(* CoDeSys 2.3.9.59 project: Pack_sorter.pro *)
(* Libraries: C:\Program Files (x86)\Common Files\CAA-Targets\Eaton Automation\V2.3.9 SP8\Lib_EC4P-200\SysLibSockets.lib, Standard.lib, SYSLIBCALLBACK.LIB, ModbusTCP.lib 14.11.23 20:05:20 *)

(* PLC configuration (modules and I/O channels)
I1 AT %IX0.0 [LocalBitInput] Input I1
I2 AT %IX0.1 [LocalBitInput] Input I2
I3 AT %IX0.2 [LocalBitInput] Input I3
I4 AT %IX0.3 [LocalBitInput] Input I4
I5 AT %IX0.4 [LocalBitInput] Input I5
I6 AT %IX0.5 [LocalBitInput] Input I6
I7 AT %IX0.6 [LocalBitInput] Input I7
I8 AT %IX0.7 [LocalBitInput] Input I8
I9 AT %IX1.0 [LocalBitInput] Input I9
I10 AT %IX1.1 [LocalBitInput] Input I10
I11 AT %IX1.2 [LocalBitInput] Input I11
I12 AT %IX1.3 [LocalBitInput] Input I12
I13 AT %IX1.4 [LocalDiagInput] Diagnostic Input I13
I14 AT %IX1.5 [LocalDiagInput] Diagnostic Input I14
I15 AT %IX1.6 [LocalDiagInput] Diagnostic Input I15
I16 AT %IX1.7 [LocalDiagInput] Diagnostic Input I16
I7_Analog AT %IW2 [LocalAnalogIn] Input I7, 10Bit, 0-10VDC
I8_Analog AT %IW4 [LocalAnalogIn] Input I8, 10Bit, 0-10VDC
I11_Analog AT %IW6 [LocalAnalogIn] Input I11, 10Bit, 0-10VDC
I12_Analog AT %IW8 [LocalAnalogIn] Input I12, 10Bit, 0-10VDC
Transistor Outputs [EC4P_TOutputs] node 0, in %IB10 out %QB0
  Q1 AT %QX0.0 [LocalBitOutput] Transistor-Output Q1
  Q2 AT %QX0.1 [LocalBitOutput] Transistor-Output Q2
  Q3 AT %QX0.2 [LocalBitOutput] Transistor-Output Q3
  Q4 AT %QX0.3 [LocalBitOutput] Transistor-Output Q4
  Q5 AT %QX0.4 [LocalBitOutput] Transistor-Output Q5
  Q6 AT %QX0.5 [LocalBitOutput] Transistor-Output Q6
  Q7 AT %QX0.6 [LocalBitOutput] Transistor-Output Q7
  Q8 AT %QX0.7 [LocalBitOutput] Transistor-Output Q8
QA1 AT %QW2 [LocalAnalogOut] 10Bit, 0-10VDC Output
No Keys [EC4P_NoKeys] node 2, in %IB10 out %QB4
No Counter [EC4P_NoCounter] node 3, in %IB10 out %QB4
Extension [EC4P_Extension] node 1, in %IB10 out %QB4
  No Extension [EC4P_NoExtension] node 0, in %IB10 out %QB4
*)

(* Global variable list: Global_Variables *)
VAR_GLOBAL
	registers :ARRAY [0..MB_MAXDATAWORDVALUE] OF WORD;
	zdalne_wejscia: ARRAY [0..4] OF WORD;
	zdalne_wyjscia: ARRAY [0..4] OF WORD;
	IZ: ARRAY [0..15] OF BOOL; (*zdalne wejscia cyfrowe*)
	QZ: ARRAY [0..15] OF BOOL; (*zdalne wyjscia cyfrowe*)
	(*valveFillSetpoint:WORD:=27648;
	valveDischargeSetpoint:WORD:=6000;
	pumpBusy:BOOL;
	systemStarted:BOOL:=FALSE;*)
END_VAR

(* Data type *)
TYPE tank :
STRUCT

	levelSensor: REAL;
	flowDischargeSensor:REAL;

	levelSetpoint:REAL:=80;
	levelLow:REAL:=60;

	valveFillAM:BOOL;
	valveFillAuto:BOOL;
	valveFillMan:BOOL;
	valveFillStart:BOOL;

	valveDischargeAM:BOOL;
	valveDischargeAuto:BOOL;
	valveDischargeMan:BOOL;
	valveDischargeStart:BOOL;

	valveFillOutput:WORD;
	valveDischargeOutput:WORD;

	FillStarted:BOOL;

	levelAlarmH:BOOL;
	levelAlarmL:BOOL;
	dischargeFlowAlarm:BOOL;
	generalFault:BOOL;

END_STRUCT
END_TYPE

(* POU PLC_PRG, LD *)
PROGRAM PLC_PRG
VAR
	max_count: INT := 100;
	SHORT_LINE: WORD := 0;
	MEDIUM_LINE: WORD := 1;
	LONG_LINE: WORD := 2;

	line_size0: WORD := 2;
	line_size1: WORD := 1;
	line_size2: WORD := 0;

	delay_emit_time: TIME := t#4s;
	ping1_on_time: TIME := t#4s;
	ping2_on_time: TIME := t#4s;
	ping3_on_time: TIME := t#4s;

	line1_time: TIME := t#6s;
	line2_time: TIME := t#6s;
	line3_time: TIME := t#5s;
	line4_time: TIME := t#6s;

	delay_ping1:  TIME := t#2s;
	delay_ping2: TIME := t#3s;
	delay_ping3: TIME := t#2s;

	destructor_time: TIME := t#5s;

	run: BOOL;
	pack_reset: BOOL;

	pack_detect: size_detect;
	new_size: WORD;
	new_pack_trig: BOOL;
	size0_count: WORD;
	size1_count: WORD;
	size2_count: WORD;

	self_emit: TON;

	pack_tracker_line1: pack_tracker;
	pack_tracker_line2: pack_tracker;
	ping1_stack_down: BOOL;
	ping2_stack_down: BOOL;

	prev_pack_line1: WORD;
	curr_pack_line1: WORD;
	prev_pack_line2: WORD;
	curr_pack_line2: WORD;

	line1_control: line_control;
	ping1_control: ping_control;
	ping1_trig: BOOL;
	ping1_size_fcn: BOOL;
	ping1_validation: ping_valid_fcn;
	ping1_enabled: BOOL;

	line2_control: line_control;
	ping2_control: ping_control1;
	ping2_trig: BOOL;
	ping2_enabled: BOOL;


	line3_control: line_control;
	ping3_control: ping_control;
	ping3_trig: BOOL;
	ping3_enable: BOOL;

	line4_control: line_control;

	destructor_line1: TOF;
	destructor_line2: TOF;
	destructor_line4: TOF;

	size0_ctu: CTU;
	size1_ctu: CTU;
	size2_ctu: CTU;
	size0: BOOL;
	size1: BOOL;
	size2: BOOL;
	emit: BOOL;
	destruct1: BOOL;
	destruct2: BOOL;
	emit_trig: F_TRIG;
	delay_emit: TOF;
	emit_tp: TOF;
	em: R_TRIG;
	p1_a, p1_b, p1_c: BOOL;
	p1_va, p1_vb, p1_vc: BOOL;
	p2_a, p2_b, p2_c: BOOL;
	p2_va, p2_vb, p2_vc: BOOL;
	p3_a, p3_b, p3_c: BOOL;
	p3_va, p3_vb, p3_vc: BOOL;

	size0_butt: button_control;
	size1_butt: button_control;
	size2_butt: button_control;
	stack_down_delay: TOF;
	prolonged_stack_down: BOOL;
	ping1_stack_delay: TOF;
	ping1_stack: BOOL;
	nowy: TP;
	init: BOOL;
	init_val: R_TRIG;
	init_trig: R_TRIG;
	default_values: R_TRIG;
END_VAR
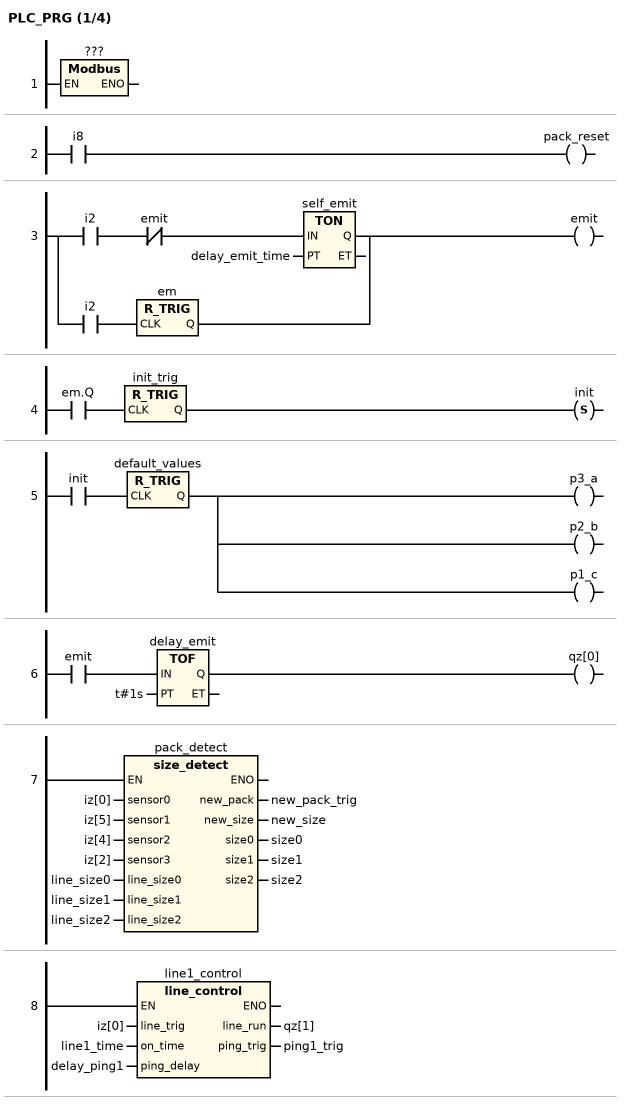
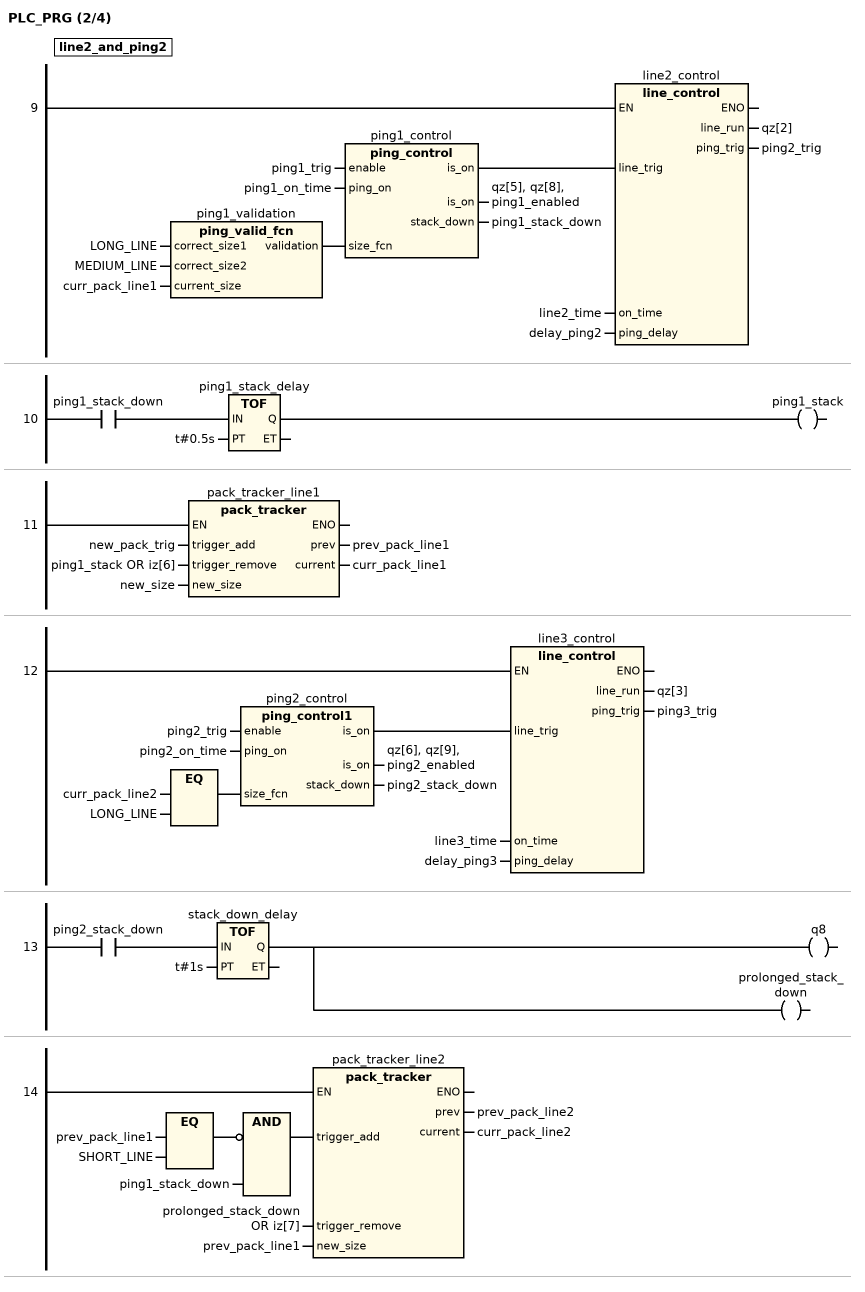
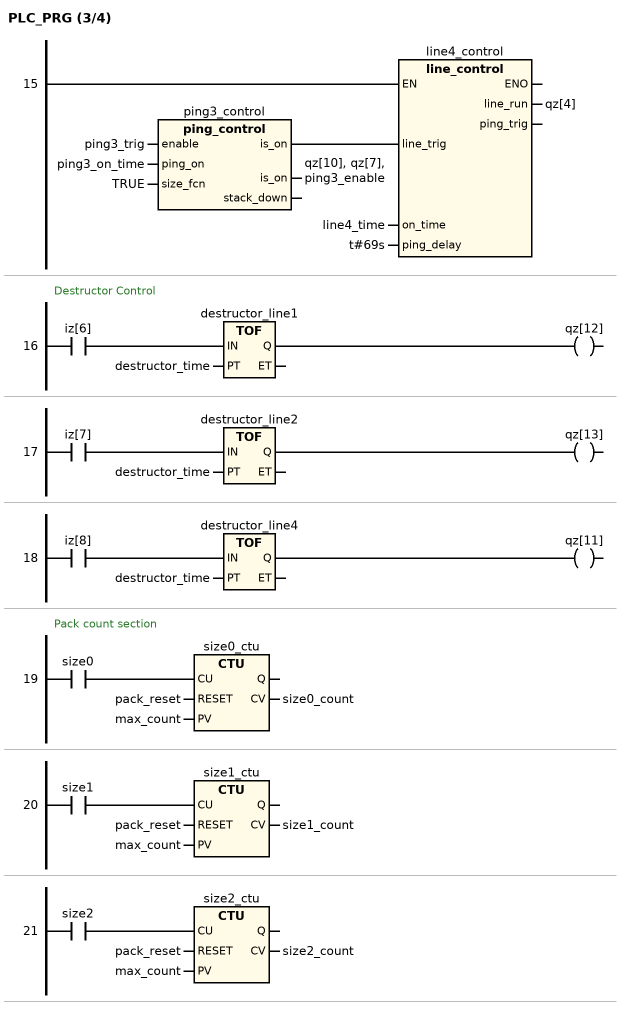
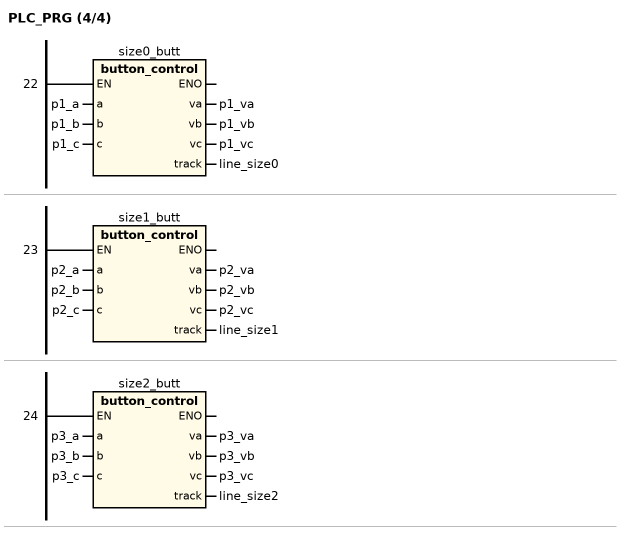
_LD_ (* Ladder Diagram *)
NETWORK 1
	*
		EN --- ???:Modbus()
NETWORK 2
	[i8] --- (pack_reset)
NETWORK 3
	{ [i2] - [/emit] - self_emit:TON(IN: *, PT: delay_emit_time) | [i2] - em:R_TRIG(CLK: *) } --- (emit)
NETWORK 4
	[em.Q] - init_trig:R_TRIG(CLK: *) --- (S init)
NETWORK 5
	[init] - default_values:R_TRIG(CLK: *) --- (p3_a) (p2_b) (p1_c)
NETWORK 6
	[emit] - delay_emit:TOF(IN: *, PT: t#1s) --- (qz[0])
NETWORK 7
	*
		EN --- pack_detect:size_detect(sensor0: iz[0], sensor1: iz[5], sensor2: iz[4], sensor3: iz[2], line_size0: line_size0, line_size1: line_size1, line_size2: line_size2, new_size => new_size, size0 => size0, size1 => size1, size2 => size2) => new_pack_trig
NETWORK 8
	*
		EN --- line1_control:line_control(line_trig: iz[0], on_time: line1_time, ping_delay: delay_ping1, ping_trig => ping1_trig) => qz[1]
NETWORK 9 line2_and_ping2:
	*
		EN --- line2_control:line_control(line_trig: <ping1_control:ping_control(enable: ping1_trig, ping_on: ping1_on_time, size_fcn: ping1_validation:ping_valid_fcn(correct_size1: LONG_LINE, correct_size2: MEDIUM_LINE, current_size: curr_pack_line1), stack_down => ping1_stack_down) => qz[5], qz[8], ping1_enabled>, on_time: line2_time, ping_delay: delay_ping2, ping_trig => ping2_trig) => qz[2]
NETWORK 10
	[ping1_stack_down] - ping1_stack_delay:TOF(IN: *, PT: t#0.5s) --- (ping1_stack)
NETWORK 11
	*
		EN --- pack_tracker_line1:pack_tracker(trigger_add: new_pack_trig, trigger_remove: ping1_stack OR iz[6], new_size: new_size, current => curr_pack_line1) => prev_pack_line1
NETWORK 12
	*
		EN --- line3_control:line_control(line_trig: <ping2_control:ping_control1(enable: ping2_trig, ping_on: ping2_on_time, size_fcn: EQ(curr_pack_line2, LONG_LINE), stack_down => ping2_stack_down) => qz[6], qz[9], ping2_enabled>, on_time: line3_time, ping_delay: delay_ping3, ping_trig => ping3_trig) => qz[3]
NETWORK 13
	[ping2_stack_down] - stack_down_delay:TOF(IN: *, PT: t#1s) --- (q8) (prolonged_stack_down)
NETWORK 14
	*
		EN --- pack_tracker_line2:pack_tracker(trigger_add: AND(NOT EQ(prev_pack_line1, SHORT_LINE), ping1_stack_down), trigger_remove: prolonged_stack_down OR iz[7], new_size: prev_pack_line1, current => curr_pack_line2) => prev_pack_line2
NETWORK 15
	*
		EN --- line4_control:line_control(line_trig: <ping3_control:ping_control(enable: ping3_trig, ping_on: ping3_on_time, size_fcn: TRUE) => qz[10], qz[7], ping3_enable>, on_time: line4_time, ping_delay: t#69s) => qz[4]
NETWORK 16 (* Destructor Control *)
	[iz[6]] - destructor_line1:TOF(IN: *, PT: destructor_time) --- (qz[12])
NETWORK 17
	[iz[7]] - destructor_line2:TOF(IN: *, PT: destructor_time) --- (qz[13])
NETWORK 18
	[iz[8]] - destructor_line4:TOF(IN: *, PT: destructor_time) --- (qz[11])
NETWORK 19 (* Pack count section *)
	[size0] - size0_ctu:CTU(CU: *, RESET: pack_reset, PV: max_count, CV => size0_count)
NETWORK 20
	[size1] - size1_ctu:CTU(CU: *, RESET: pack_reset, PV: max_count, CV => size1_count)
NETWORK 21
	[size2] - size2_ctu:CTU(CU: *, RESET: pack_reset, PV: max_count, CV => size2_count)
NETWORK 22
	*
		EN --- size0_butt:button_control(a: p1_a, b: p1_b, c: p1_c, vb => p1_vb, vc => p1_vc, track => line_size0) => p1_va
NETWORK 23
	*
		EN --- size1_butt:button_control(a: p2_a, b: p2_b, c: p2_c, vb => p2_vb, vc => p2_vc, track => line_size1) => p2_va
NETWORK 24
	*
		EN --- size2_butt:button_control(a: p3_a, b: p3_b, c: p3_c, vb => p3_vb, vc => p3_vc, track => line_size2) => p3_va
_END_LD_
(* the same logic as Structured Text *)
(* Network 1: see the listing above *)
(* Network 2 *)
pack_reset := i8;
(* Network 3 *)
self_emit(IN := i2 AND NOT emit, PT := delay_emit_time);
em(CLK := i2);
emit := self_emit.Q OR em.Q;
(* Network 4 *)
init_trig(CLK := em.Q);
IF init_trig.Q THEN init := TRUE; END_IF;
(* Network 5 *)
default_values(CLK := init);
p3_a := default_values.Q;
p2_b := default_values.Q;
p1_c := default_values.Q;
(* Network 6 *)
delay_emit(IN := emit, PT := t#1s);
qz[0] := delay_emit.Q;
(* Network 7 *)
pack_detect(sensor0 := iz[0], sensor1 := iz[5], sensor2 := iz[4], sensor3 := iz[2], line_size0 := line_size0, line_size1 := line_size1, line_size2 := line_size2);
new_size := pack_detect.new_size;
size0 := pack_detect.size0;
size1 := pack_detect.size1;
size2 := pack_detect.size2;
new_pack_trig := pack_detect.new_pack;
(* Network 8 *)
line1_control(line_trig := iz[0], on_time := line1_time, ping_delay := delay_ping1);
ping1_trig := line1_control.ping_trig;
qz[1] := line1_control.line_run;
(* Network 9: see the listing above *)
(* Network 10 *)
ping1_stack_delay(IN := ping1_stack_down, PT := t#0.5s);
ping1_stack := ping1_stack_delay.Q;
(* Network 11 *)
pack_tracker_line1(trigger_add := new_pack_trig, trigger_remove := ping1_stack OR iz[6], new_size := new_size);
curr_pack_line1 := pack_tracker_line1.current;
prev_pack_line1 := pack_tracker_line1.prev;
(* Network 12: see the listing above *)
(* Network 13 *)
stack_down_delay(IN := ping2_stack_down, PT := t#1s);
q8 := stack_down_delay.Q;
prolonged_stack_down := stack_down_delay.Q;
(* Network 14 *)
pack_tracker_line2(trigger_add := NOT (prev_pack_line1 = SHORT_LINE) AND ping1_stack_down, trigger_remove := prolonged_stack_down OR iz[7], new_size := prev_pack_line1);
curr_pack_line2 := pack_tracker_line2.current;
prev_pack_line2 := pack_tracker_line2.prev;
(* Network 15: see the listing above *)
(* Network 16 *)
destructor_line1(IN := iz[6], PT := destructor_time);
qz[12] := destructor_line1.Q;
(* Network 17 *)
destructor_line2(IN := iz[7], PT := destructor_time);
qz[13] := destructor_line2.Q;
(* Network 18 *)
destructor_line4(IN := iz[8], PT := destructor_time);
qz[11] := destructor_line4.Q;
(* Network 19 *)
size0_ctu(CU := size0, RESET := pack_reset, PV := max_count);
size0_count := size0_ctu.CV;
(* Network 20 *)
size1_ctu(CU := size1, RESET := pack_reset, PV := max_count);
size1_count := size1_ctu.CV;
(* Network 21 *)
size2_ctu(CU := size2, RESET := pack_reset, PV := max_count);
size2_count := size2_ctu.CV;
(* Network 22 *)
size0_butt(a := p1_a, b := p1_b, c := p1_c);
p1_vb := size0_butt.vb;
p1_vc := size0_butt.vc;
line_size0 := size0_butt.track;
p1_va := size0_butt.va;
(* Network 23 *)
size1_butt(a := p2_a, b := p2_b, c := p2_c);
p2_vb := size1_butt.vb;
p2_vc := size1_butt.vc;
line_size1 := size1_butt.track;
p2_va := size1_butt.va;
(* Network 24 *)
size2_butt(a := p3_a, b := p3_b, c := p3_c);
p3_vb := size2_butt.vb;
p3_vc := size2_butt.vc;
line_size2 := size2_butt.track;
p3_va := size2_butt.va;
END_PROGRAM

(* POU size_detect, ST *)
FUNCTION_BLOCK size_detect
VAR_INPUT
	(*  iz[0] - s0; iz[5] - s1; iz[4]; s2-  iz[2] *)
	sensor0, sensor1, sensor2, sensor3: BOOL;
	line_size0, line_size1, line_size2: WORD;
END_VAR
VAR_OUTPUT
	new_pack: BOOL;
	new_size: WORD;
	size0, size1, size2: BOOL;
END_VAR
VAR
	size0_trg, reset_trg, size2_trg: R_TRIG;
	size0_det: BOOL := FALSE;
END_VAR
size0_trg(CLK := sensor0);
size2_trg(CLK := sensor2);
reset_trg(CLK := sensor3);

IF size0_trg.Q AND sensor1 THEN
	new_size := line_size0;
	size0  := TRUE;
	size1 := FALSE;
	size2 := FALSE;
	size0_det := TRUE;

	new_pack := TRUE;
ELSIF size2_trg.Q AND NOT size0_det  THEN
	IF sensor3 THEN
		new_size := line_size1;
		size1  := TRUE;
		size0 := FALSE;
		size2 := FALSE;
		size0_det := FALSE;

		new_pack := TRUE;
	ELSE
		new_size := line_size2;
		size2  := TRUE;
		size1 := FALSE;
		size0 := FALSE;
		size0_det := FALSE;

		new_pack := TRUE;
	END_IF;
ELSIF reset_trg.Q THEN
	size0_det := FALSE;
	size1 := FALSE;
	size1 := FALSE;
	size0 := FALSE;
ELSE
	new_pack := FALSE;
	size1 := FALSE;
	size1 := FALSE;
	size0 := FALSE;
END_IF;
END_FUNCTION_BLOCK

(* POU pack_tracker, ST *)
FUNCTION_BLOCK pack_tracker
VAR_INPUT
	trigger_add: BOOL;
	trigger_remove: BOOL;
	new_size: WORD;
END_VAR
VAR_OUTPUT
	prev: WORD := 255;
	current: WORD := 255;
END_VAR
VAR
	stack_size: INT := 6;
	stack : ARRAY [1..6] OF WORD;
	stack_init: BOOL := TRUE;

	stack_up_trig: R_TRIG;
	stack_down_trig: R_TRIG;
	i: INT;
END_VAR
stack_up_trig(CLK := trigger_add);
stack_down_trig(CLK := trigger_remove);

IF stack_init THEN
	FOR i :=1 TO stack_size DO
		stack[i] := 255;
	END_FOR;
	stack_init := FALSE;
END_IF;

IF stack_down_trig.Q THEN
	prev := stack[1];
	FOR i := 1 TO stack_size-1 DO
		IF stack[i] = 255 THEN
			EXIT;
		END_IF;

		stack[i] := stack[i+1];
	END_FOR;
	current := stack[1];
END_IF;

IF stack_up_trig.Q THEN
	FOR i := 1	 TO stack_size-1 DO
		IF stack[i] = 255 THEN
			stack[i] := new_size;
			IF i = 1 THEN
				current := new_size;
			END_IF;

			EXIT;
		END_IF;
	END_FOR;
END_IF;
END_FUNCTION_BLOCK

(* POU line_control, LD *)
FUNCTION_BLOCK line_control
VAR_INPUT
	line_trig: BOOL;
	on_time: TIME;
	ping_delay: TIME;
END_VAR
VAR_OUTPUT
	line_run: BOOL;
	ping_trig: BOOL;
END_VAR
VAR
	line_enable_trig: R_TRIG;
	line_on: BOOL;
	ping_timer: TON;
	line_run_timer: TOF;
	ping_off: BOOL;
	timing_error: BOOL;

	ping_delay_timer: TP;
	ping_trigger: F_TRIG;
END_VAR
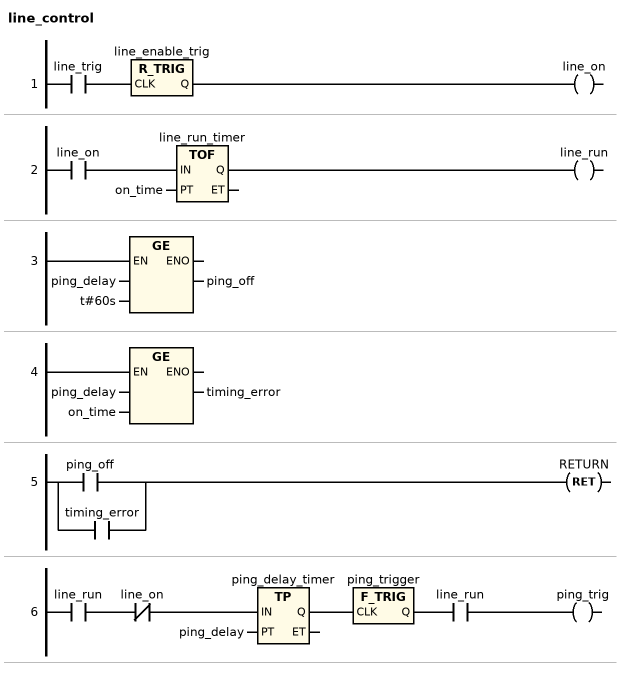
_LD_ (* Ladder Diagram *)
NETWORK 1
	[line_trig] - line_enable_trig:R_TRIG(CLK: *) --- (line_on)
NETWORK 2
	[line_on] - line_run_timer:TOF(IN: *, PT: on_time) --- (line_run)
NETWORK 3
	*
		EN --- GE(ping_delay, t#60s) => ping_off
NETWORK 4
	*
		EN --- GE(ping_delay, on_time) => timing_error
NETWORK 5
	{ [ping_off] | [timing_error] } --- <RETURN>
NETWORK 6
	[line_run] - [/line_on] - ping_delay_timer:TP(IN: *, PT: ping_delay) - ping_trigger:F_TRIG(CLK: *) - [line_run] --- (ping_trig)
_END_LD_
(* the same logic as Structured Text *)
(* Network 1 *)
line_enable_trig(CLK := line_trig);
line_on := line_enable_trig.Q;
(* Network 2 *)
line_run_timer(IN := line_on, PT := on_time);
line_run := line_run_timer.Q;
(* Network 3 *)
ping_off := ping_delay >= t#60s;
(* Network 4 *)
timing_error := ping_delay >= on_time;
(* Network 5 *)
IF ping_off OR timing_error THEN RETURN; END_IF;
(* Network 6 *)
ping_delay_timer(IN := line_run AND NOT line_on, PT := ping_delay);
ping_trigger(CLK := ping_delay_timer.Q);
ping_trig := ping_trigger.Q AND line_run;
END_FUNCTION_BLOCK

(* POU ping_control, LD *)
FUNCTION_BLOCK ping_control
VAR_INPUT
	enable: BOOL;
	ping_on: TIME;
	size_fcn: BOOL;
END_VAR
VAR_OUTPUT
	is_on: BOOL;
	stack_down: BOOL;
END_VAR
VAR
	start_time: R_TRIG;
	turn_on: BOOL;
	delay_timer: TOF;
	size: BOOL;
	helper_counter: CTUD;
	odd_pack: BOOL;
	even_pack: BOOL;
	even_pack_timer: TOF;
	odd_pack_timer: TOF;
	stack_down_trig: F_TRIG;
	stack_down_odd: BOOL;
	stack_down_odd_trig: F_TRIG;
	stack_down_even_trig: F_TRIG;
	stack_down_even: BOOL;
	odd_timer_trig: F_TRIG;
	even_timer_trig: F_TRIG;
	cu_en: BOOL;
	cd_en: BOOL;
	od_tp: TP;
	ev_tp: TP;
END_VAR
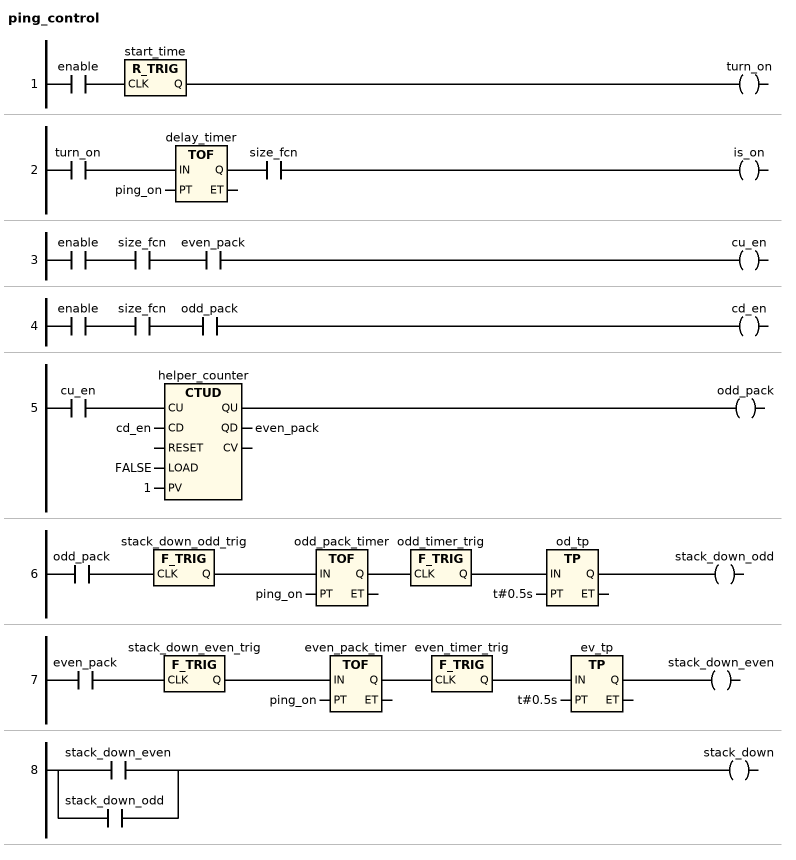
_LD_ (* Ladder Diagram *)
NETWORK 1
	[enable] - start_time:R_TRIG(CLK: *) --- (turn_on)
NETWORK 2
	[turn_on] - delay_timer:TOF(IN: *, PT: ping_on) - [size_fcn] --- (is_on)
NETWORK 3
	[enable] - [size_fcn] - [even_pack] --- (cu_en)
NETWORK 4
	[enable] - [size_fcn] - [odd_pack] --- (cd_en)
NETWORK 5
	[cu_en] - helper_counter:CTUD(CU: *, CD: cd_en, RESET: , LOAD: FALSE, PV: 1, QD => even_pack) --- (odd_pack)
NETWORK 6
	[odd_pack] - stack_down_odd_trig:F_TRIG(CLK: *) - odd_pack_timer:TOF(IN: *, PT: ping_on) - odd_timer_trig:F_TRIG(CLK: *) - od_tp:TP(IN: *, PT: t#0.5s) --- (stack_down_odd)
NETWORK 7
	[even_pack] - stack_down_even_trig:F_TRIG(CLK: *) - even_pack_timer:TOF(IN: *, PT: ping_on) - even_timer_trig:F_TRIG(CLK: *) - ev_tp:TP(IN: *, PT: t#0.5s) --- (stack_down_even)
NETWORK 8
	{ [stack_down_even] | [stack_down_odd] } --- (stack_down)
_END_LD_
(* the same logic as Structured Text *)
(* Network 1 *)
start_time(CLK := enable);
turn_on := start_time.Q;
(* Network 2 *)
delay_timer(IN := turn_on, PT := ping_on);
is_on := delay_timer.Q AND size_fcn;
(* Network 3 *)
cu_en := enable AND size_fcn AND even_pack;
(* Network 4 *)
cd_en := enable AND size_fcn AND odd_pack;
(* Network 5: see the listing above *)
(* Network 6 *)
stack_down_odd_trig(CLK := odd_pack);
odd_pack_timer(IN := stack_down_odd_trig.Q, PT := ping_on);
odd_timer_trig(CLK := odd_pack_timer.Q);
od_tp(IN := odd_timer_trig.Q, PT := t#0.5s);
stack_down_odd := od_tp.Q;
(* Network 7 *)
stack_down_even_trig(CLK := even_pack);
even_pack_timer(IN := stack_down_even_trig.Q, PT := ping_on);
even_timer_trig(CLK := even_pack_timer.Q);
ev_tp(IN := even_timer_trig.Q, PT := t#0.5s);
stack_down_even := ev_tp.Q;
(* Network 8 *)
stack_down := stack_down_even OR stack_down_odd;
END_FUNCTION_BLOCK

(* POU ping_valid_fcn, LD *)
FUNCTION_BLOCK ping_valid_fcn
VAR_INPUT
	correct_size1, correct_size2: WORD;
	current_size: WORD;
END_VAR
VAR_OUTPUT
	validation: BOOL;
END_VAR
VAR
END_VAR
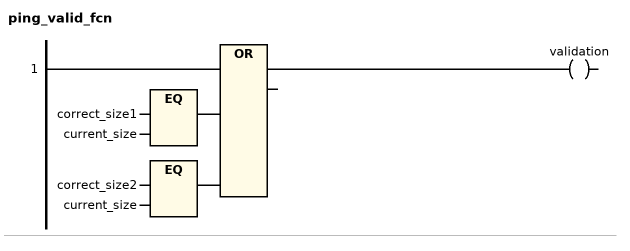
_LD_ (* Ladder Diagram *)
NETWORK 1
	OR(EQ(correct_size1, current_size), EQ(correct_size2, current_size)) --- (validation)
_END_LD_
END_FUNCTION_BLOCK

(* POU ping_control1, LD *)
FUNCTION_BLOCK ping_control1
VAR_INPUT
	enable: BOOL;
	ping_on: TIME;
	size_fcn: BOOL;
END_VAR
VAR_OUTPUT
	is_on: BOOL;
	stack_down: BOOL;
END_VAR
VAR
	start_time: R_TRIG;
	turn_on: BOOL;
	delay_timer: TOF;
	size: BOOL;
	helper_counter: CTUD;
	odd_pack: BOOL;
	even_pack: BOOL;
	even_pack_timer: TOF;
	odd_pack_timer: TOF;
	stack_down_trig: F_TRIG;
	stack_down_odd: BOOL;
	stack_down_odd_trig: F_TRIG;
	stack_down_even_trig: F_TRIG;
	stack_down_even: BOOL;
	odd_timer_trig: F_TRIG;
	even_timer_trig: F_TRIG;
	cu_en: BOOL;
	cd_en: BOOL;
	init: BOOL;
	init_trig: R_TRIG;
	od: TP;
	ev: TP;
END_VAR
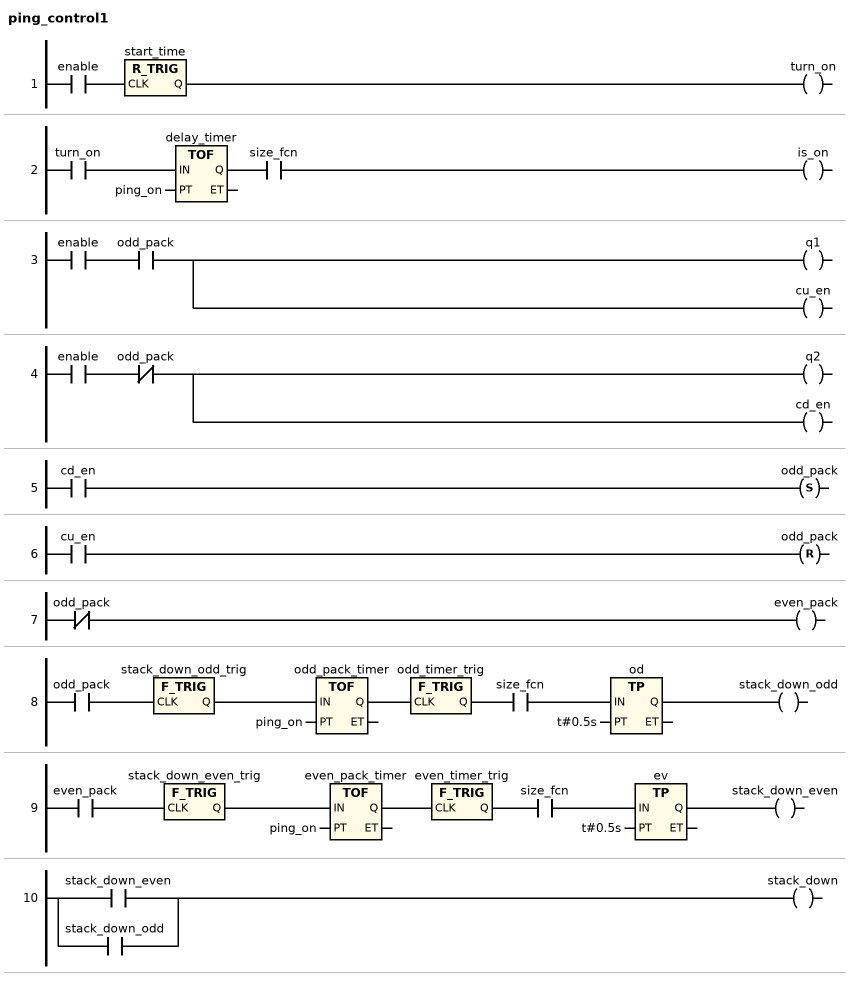
_LD_ (* Ladder Diagram *)
NETWORK 1
	[enable] - start_time:R_TRIG(CLK: *) --- (turn_on)
NETWORK 2
	[turn_on] - delay_timer:TOF(IN: *, PT: ping_on) - [size_fcn] --- (is_on)
NETWORK 3
	[enable] - [odd_pack] --- (q1) (cu_en)
NETWORK 4
	[enable] - [/odd_pack] --- (q2) (cd_en)
NETWORK 5
	[cd_en] --- (S odd_pack)
NETWORK 6
	[cu_en] --- (R odd_pack)
NETWORK 7
	[/odd_pack] --- (even_pack)
NETWORK 8
	[odd_pack] - stack_down_odd_trig:F_TRIG(CLK: *) - odd_pack_timer:TOF(IN: *, PT: ping_on) - odd_timer_trig:F_TRIG(CLK: *) - [size_fcn] - od:TP(IN: *, PT: t#0.5s) --- (stack_down_odd)
NETWORK 9
	[even_pack] - stack_down_even_trig:F_TRIG(CLK: *) - even_pack_timer:TOF(IN: *, PT: ping_on) - even_timer_trig:F_TRIG(CLK: *) - [size_fcn] - ev:TP(IN: *, PT: t#0.5s) --- (stack_down_even)
NETWORK 10
	{ [stack_down_even] | [stack_down_odd] } --- (stack_down)
_END_LD_
(* the same logic as Structured Text *)
(* Network 1 *)
start_time(CLK := enable);
turn_on := start_time.Q;
(* Network 2 *)
delay_timer(IN := turn_on, PT := ping_on);
is_on := delay_timer.Q AND size_fcn;
(* Network 3 *)
q1 := enable AND odd_pack;
cu_en := q1;
(* Network 4 *)
q2 := enable AND NOT odd_pack;
cd_en := q2;
(* Network 5 *)
IF cd_en THEN odd_pack := TRUE; END_IF;
(* Network 6 *)
IF cu_en THEN odd_pack := FALSE; END_IF;
(* Network 7 *)
even_pack := NOT odd_pack;
(* Network 8 *)
stack_down_odd_trig(CLK := odd_pack);
odd_pack_timer(IN := stack_down_odd_trig.Q, PT := ping_on);
odd_timer_trig(CLK := odd_pack_timer.Q);
od(IN := odd_timer_trig.Q AND size_fcn, PT := t#0.5s);
stack_down_odd := od.Q;
(* Network 9 *)
stack_down_even_trig(CLK := even_pack);
even_pack_timer(IN := stack_down_even_trig.Q, PT := ping_on);
even_timer_trig(CLK := even_pack_timer.Q);
ev(IN := even_timer_trig.Q AND size_fcn, PT := t#0.5s);
stack_down_even := ev.Q;
(* Network 10 *)
stack_down := stack_down_even OR stack_down_odd;
END_FUNCTION_BLOCK

(* POU button_control, LD *)
FUNCTION_BLOCK button_control
VAR_INPUT
	a, b, c : BOOL;
END_VAR
VAR_OUTPUT
	va, vb, vc: BOOL;
	track: WORD;
END_VAR
VAR
END_VAR
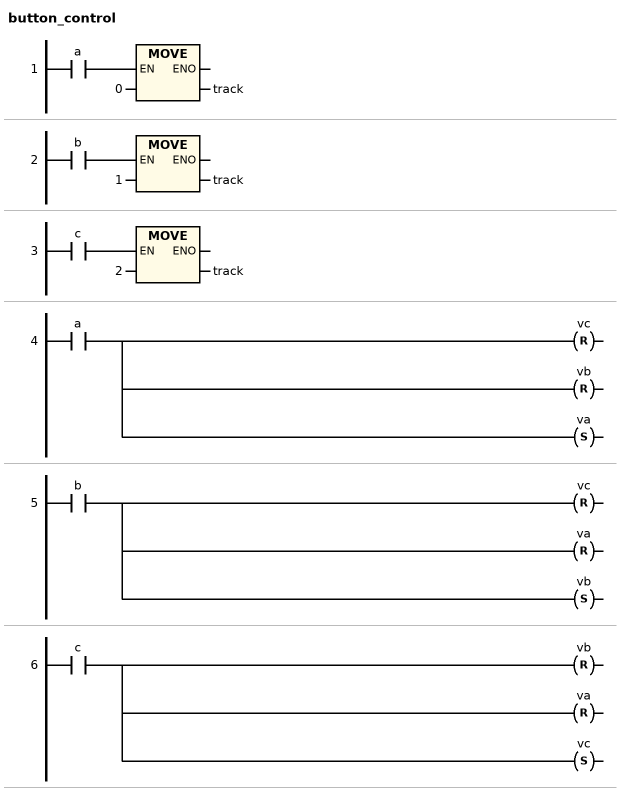
_LD_ (* Ladder Diagram *)
NETWORK 1
	[a]
		EN --- MOVE(0) => track
NETWORK 2
	[b]
		EN --- MOVE(1) => track
NETWORK 3
	[c]
		EN --- MOVE(2) => track
NETWORK 4
	[a] --- (R vc) (R vb) (S va)
NETWORK 5
	[b] --- (R vc) (R va) (S vb)
NETWORK 6
	[c] --- (R vb) (R va) (S vc)
_END_LD_
(* the same logic as Structured Text *)
(* Network 1 *)
IF a THEN
	track := 0;
END_IF;
(* Network 2 *)
IF b THEN
	track := 1;
END_IF;
(* Network 3 *)
IF c THEN
	track := 2;
END_IF;
(* Network 4 *)
IF a THEN vc := FALSE; vb := FALSE; va := TRUE; END_IF;
(* Network 5 *)
IF b THEN vc := FALSE; va := FALSE; vb := TRUE; END_IF;
(* Network 6 *)
IF c THEN vb := FALSE; va := FALSE; vc := TRUE; END_IF;
END_FUNCTION_BLOCK

(* POU Modbus, ST *)
PROGRAM Modbus

VAR
	modbusError: WORD;
	modbusTCP_server:FB_serverModbusTCP;
	FB_mapInputRegister:FB_mapInputRegister;
	FB_mapOutputRegister:FB_mapOutputRegister;
	FB_startSystem:FB_startSystem;
	FB_liveBitMonitor:FB_liveBitMonitor;
	startDischarge: BOOL;
	deviceFault: BOOL;
	faultAcknowledge: BOOL;
	i:SINT;
	stopLight: BOOL;
	voltageLight: BOOL;
	liveBitBitInput: BOOL;
	liveBitBitOutput: BOOL;
	modbusTimeoutError: BOOL;
	copy_zdalne1: copy_zdalne;
END_VAR
(* Modbus server FB *)
modbusTCP_server(ServerID:=255 , ServerPort:=502 , LastError=>modbusError);

(* Mapping input registers to variables *)
copy_zdalne1(EN:=TRUE);

(*FB_mapInputRegister(
	inputHoldingRegister:=registers[0] ,
	bit0=> Q1,
	bit1=> Q2,
	bit2=> Q3,
	bit3=> Q4,
	bit4=> Q5,
	bit5=> Q6 ,
	bit6=> Q7,
	bit7=> Q8,
	bit8=> ,
	bit9=> ,
	bit10=> ,
	bit11=> ,
	bit12=> ,
	bit13=> ,
	bit14=> ,
	bit15=> liveBitBitInput);
*)
FB_mapInputRegister(
	inputHoldingRegister:=registers[0] ,
	bit0=> IZ[0],
	bit1=> IZ[1],
	bit2=> IZ[2],
	bit3=> IZ[3],
	bit4=> IZ[4],
	bit5=> IZ[5] ,
	bit6=> IZ[6],
	bit7=> IZ[7],
	bit8=> IZ[8],
	bit9=> IZ[9],
	bit10=> IZ[10],
	bit11=> IZ[11],
	bit12=> IZ[12],
	bit13=> IZ[13],
	bit14=> IZ[14],
	bit15=> IZ[15]);

(* Modbus liveBit *)
FB_liveBitMonitor(liveBitInput:=liveBitBitInput , liveBitOutput=>liveBitBitOutput , liveBitError=> modbusTimeoutError);

(* Process faults *)


(* Process control *)



(* Fault acknowledge *)



(* Map variables to output registers *)

FB_mapOutputRegister(
	bit0:= QZ[0],
	bit1:= QZ[1],
	bit2:= QZ[2],
	bit3:= QZ[3],
	bit4:= QZ[4],
	bit5:= QZ[5],
	bit6:= QZ[6],
	bit7:= QZ[7],
	bit8:= QZ[8],
	bit9:= QZ[9],
	bit10:= QZ[10],
	bit11:= QZ[11],
	bit12:= QZ[12],
	bit13:= QZ[13],
	bit14:= QZ[14],
	bit15:= QZ[15],
	outputHoldingRegister=>registers[60] );
(*FB_mapOutputRegister(
	bit0:= I1,
	bit1:= I2,
	bit2:= I3,
	bit3:= I4,
	bit4:= I5,
	bit5:= I6,
	bit6:= I7,
	bit7:= I8,
	bit8:= I9,
	bit9:= I10,
	bit10:= I11,
	bit11:= I12,
	bit12:= ,
	bit13:= ,
	bit14:= ,
	bit15:= ,
	outputHoldingRegister=>registers[60] );
*)

qa1:= REGISTERS[1];
registers[61]:=i7_analog;
registers[62]:=i8_analog;

registers[63]:=i11_analog;
registers[64]:=i12_analog;

registers[65]:=0;
registers[66]:=0;

registers[67]:=0;
registers[68]:=0;

registers[119] := registers[119]+1;
END_PROGRAM

(* POU FBs/FB_serverModbusTCP, ST *)
FUNCTION_BLOCK FB_serverModbusTCP
VAR_INPUT
	ServerID:BYTE;
	ServerPort:INT;
END_VAR
VAR_OUTPUT
	LastError:INT;
END_VAR
VAR
	SlaveSetup:MBS_Setup;
	SlavePoll:MBS_Poll;
	SlaveAnswer:MBS_Answer;
	step: USINT :=0;
	i: INT;
END_VAR
CASE step OF
0:	(*Initialisation*)

	SlaveSetup.bUnitIdentifier := ServerID;
	MBS_AcceptAllSubunitIds := TRUE;

	SlaveSetup.wDefaultPort :=ServerPort;
	SlaveSetup.xDefaultPortActive:=TRUE;
	SlaveSetup.xAdditionalPortActive:=FALSE;

	SlaveSetup.xSecureMode:=FALSE;			(*If TRUE only preset IPs are accepted*)
	SlaveSetup.tTimeout:=T#1m;					(*Timeout if no communication with slave established*)
	SlaveSetup(xStrobe:=TRUE);					(*Strobe starts function*)
	IF SlaveSetup.xBusy = FALSE THEN
		SlaveSetup(xstrobe := FALSE);			(*provides falling edge*)
		step := 1 ;
	END_IF;
1:
	SlavePoll(xStrobe:=TRUE);					(*waiting for incomming master commands*)
		IF NOT SlavePoll.xBusy THEN
			step:=2;							(*hint: step 1 & 2 could be merged to accelerate slave handling, if needed*)
			SlavePoll(xStrobe:=FALSE);			(*provides falling edge*)
		END_IF;

2:
	step:= 1;

	IF  SlavePoll.xAvailable = TRUE  THEN

		IF SlavePoll.iErrorCode <> 0 THEN
			LastError := SlavePoll.iErrorCode;									(* provided for error treatment *)
		END_IF;

		CASE SlavePoll.bFunctionCode OF										(* connect accepted pollparameters with answerparameters *)
			16:
				slaveanswer.bFunctionCode:=slavepoll.bFunctionCode;
				slaveanswer.wCount:=slavepoll.wCount;
				slaveanswer.wOffset:=slavepoll.wOffset;
				FOR i := 0 TO slaveanswer.wCount-1 BY 1 DO
					registers[slaveanswer.woffset+i] := slavepoll.warData[i];		(*Write to Data-array*)
				END_FOR;
				slaveanswer.wardata := slavepoll.warData;
			4:
				slaveanswer.bFunctionCode:=slavepoll.bFunctionCode;
				slaveanswer.wCount:=slavepoll.wCount;
				slaveanswer.wOffset:=slavepoll.wOffset;
				FOR i:= 0 TO slaveanswer.wCount-1 BY 1 DO
					slaveanswer.warData[i]:=registers[slavepoll.woffset+i];			(*Read from Data-array*)
				END_FOR
		END_CASE;

		slaveanswer();	(*When Data ready, send answer*)

	END_IF;
END_CASE;
END_FUNCTION_BLOCK

(* POU FBs/FB_mapInputRegister, ST *)
FUNCTION_BLOCK FB_mapInputRegister
VAR_INPUT
	inputHoldingRegister : WORD;
END_VAR
VAR_OUTPUT
	bit0 : BOOL;
	bit1 : BOOL;
	bit2 : BOOL;
	bit3 : BOOL;
	bit4 : BOOL;
	bit5 : BOOL;
	bit6 : BOOL;
	bit7 : BOOL;
	bit8 : BOOL;
	bit9 : BOOL;
	bit10 : BOOL;
	bit11 : BOOL;
	bit12 : BOOL;
	bit13 : BOOL;
	bit14 : BOOL;
	bit15 : BOOL;
END_VAR
VAR
END_VAR
bit0 :=inputHoldingRegister.0;
bit1 :=inputHoldingRegister.1;
bit2 :=inputHoldingRegister.2;
bit3 :=inputHoldingRegister.3;
bit4 :=inputHoldingRegister.4;
bit5 :=inputHoldingRegister.5;
bit6 :=inputHoldingRegister.6;
bit7 :=inputHoldingRegister.7;
bit8 :=inputHoldingRegister.8;
bit9 :=inputHoldingRegister.9;
bit10 :=inputHoldingRegister.10;
bit11 :=inputHoldingRegister.11;
bit12 :=inputHoldingRegister.12;
bit13 :=inputHoldingRegister.13;
bit14 :=inputHoldingRegister.14;
bit15 :=inputHoldingRegister.15;
END_FUNCTION_BLOCK

(* POU FBs/FB_mapOutputRegister, ST *)
FUNCTION_BLOCK FB_mapOutputRegister
VAR_INPUT
	bit0 : BOOL;
	bit1 : BOOL;
	bit2 : BOOL;
	bit3 : BOOL;
	bit4 : BOOL;
	bit5 : BOOL;
	bit6 : BOOL;
	bit7 : BOOL;
	bit8 : BOOL;
	bit9 : BOOL;
	bit10 : BOOL;
	bit11 : BOOL;
	bit12 : BOOL;
	bit13 : BOOL;
	bit14 : BOOL;
	bit15 : BOOL;
END_VAR
VAR_OUTPUT
	outputHoldingRegister : WORD;
END_VAR
VAR
END_VAR
outputHoldingRegister.0:=bit0;
outputHoldingRegister.1:=bit1;
outputHoldingRegister.2:=bit2;
outputHoldingRegister.3:=bit3;
outputHoldingRegister.4:=bit4;
outputHoldingRegister.5:=bit5;
outputHoldingRegister.6:=bit6;
outputHoldingRegister.7:=bit7;
outputHoldingRegister.8:=bit8;
outputHoldingRegister.9:=bit9;
outputHoldingRegister.10:=bit10;
outputHoldingRegister.11:=bit11;
outputHoldingRegister.12:=bit12;
outputHoldingRegister.13:=bit13;
outputHoldingRegister.14:=bit14;
outputHoldingRegister.15:=bit15;
END_FUNCTION_BLOCK

(* POU FBs/FB_startSystem, LD *)
FUNCTION_BLOCK FB_startSystem
VAR_INPUT
	start:BOOL;
	stop:BOOL;
	safety:BOOL;
	reset:BOOL;
	fault:BOOL;
END_VAR
VAR_OUTPUT
	systemStarted:BOOL;
	systemStopLight: BOOL;
	safetyRS: BOOL:=TRUE;
END_VAR
VAR
	TOF_BLINK: TOF;
	TON_BLINK: TON;

END_VAR
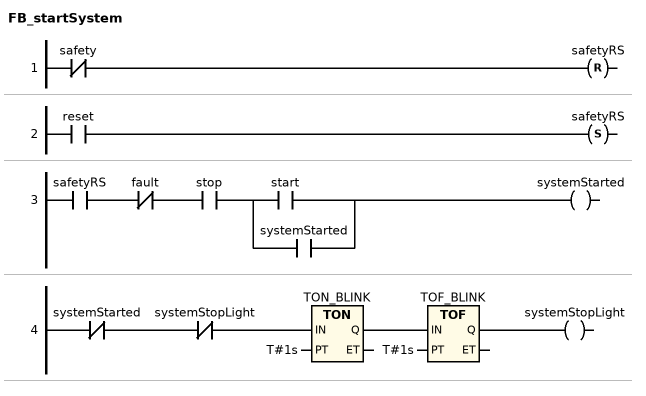
_LD_ (* Ladder Diagram *)
NETWORK 1
	[/safety] --- (R safetyRS)
NETWORK 2
	[reset] --- (S safetyRS)
NETWORK 3
	[safetyRS] - [/fault] - [stop] - { [start] | [systemStarted] } --- (systemStarted)
NETWORK 4
	[/systemStarted] - [/systemStopLight] - TON_BLINK:TON(IN: *, PT: T#1s) - TOF_BLINK:TOF(IN: *, PT: T#1s) --- (systemStopLight)
_END_LD_
(* the same logic as Structured Text *)
(* Network 1 *)
IF NOT safety THEN safetyRS := FALSE; END_IF;
(* Network 2 *)
IF reset THEN safetyRS := TRUE; END_IF;
(* Network 3 *)
systemStarted := safetyRS AND NOT fault AND stop AND (start OR systemStarted);
(* Network 4 *)
TON_BLINK(IN := NOT systemStarted AND NOT systemStopLight, PT := T#1s);
TOF_BLINK(IN := TON_BLINK.Q, PT := T#1s);
systemStopLight := TOF_BLINK.Q;
END_FUNCTION_BLOCK

(* POU FBs/FB_liveBitMonitor, ST *)
FUNCTION_BLOCK FB_liveBitMonitor
VAR_INPUT
	liveBitInput:BOOL;
END_VAR
VAR_OUTPUT
	liveBitOutput:BOOL;
	liveBitError:BOOL;
END_VAR
VAR
	inputR_TRIG: R_TRIG;
	liveBitTON: TON;
END_VAR
inputR_TRIG(CLK:=liveBitInput , Q=> );

liveBitTON(IN:= NOT inputR_TRIG.Q , PT:= T#3s , Q=> , ET=> );

IF liveBitTON.Q THEN
	liveBitError:=TRUE;
END_IF;
IF inputR_TRIG.Q THEN
	liveBitError:=FALSE;
END_IF

liveBitOutput := liveBitInput;
END_FUNCTION_BLOCK

(* POU FBs/copy_zdalne, ST *)
FUNCTION_BLOCK copy_zdalne
VAR_INPUT
	EN:BOOL;
END_VAR
VAR_OUTPUT
END_VAR
VAR
	k:INT;
END_VAR
(*FOR k:=0 TO 15 BY 1 DO
	zdalne_wyjscia[0].k := QZ[k];
END_FOR*)
IF EN THEN
zdalne_wyjscia[0].0 := QZ[0];
zdalne_wyjscia[0].1 := QZ[1];
zdalne_wyjscia[0].2 := QZ[2];
zdalne_wyjscia[0].3 := QZ[3];
zdalne_wyjscia[0].4 := QZ[4];
zdalne_wyjscia[0].5 := QZ[5];
zdalne_wyjscia[0].6 := QZ[6];
zdalne_wyjscia[0].7 := QZ[7];
zdalne_wyjscia[0].8 := QZ[8];
zdalne_wyjscia[0].9 := QZ[9];
zdalne_wyjscia[0].10 := QZ[10];
zdalne_wyjscia[0].11 := QZ[11];
zdalne_wyjscia[0].12 := QZ[12];
zdalne_wyjscia[0].13 := QZ[13];
zdalne_wyjscia[0].14 := QZ[14];
zdalne_wyjscia[0].15 := QZ[15];

registers[60]:=zdalne_wyjscia[0];
registers[61]:=zdalne_wyjscia[1];
registers[62]:=zdalne_wyjscia[2];
registers[63]:=zdalne_wyjscia[3];
registers[64]:=zdalne_wyjscia[4];

zdalne_wejscia[0]:=registers[0];
zdalne_wejscia[1]:=registers[1];
zdalne_wejscia[2]:=registers[2];
zdalne_wejscia[3]:=registers[3];
zdalne_wejscia[4]:=registers[4];

IZ[0] := zdalne_wejscia[0].0;
IZ[1] := zdalne_wejscia[0].1;
IZ[2] := zdalne_wejscia[0].2;
IZ[3] := zdalne_wejscia[0].3;
IZ[4] := zdalne_wejscia[0].4;
IZ[5] := zdalne_wejscia[0].5;
IZ[6] := zdalne_wejscia[0].6;
IZ[7] := zdalne_wejscia[0].7;
IZ[8] := zdalne_wejscia[0].8;
IZ[9] := zdalne_wejscia[0].9;
IZ[10] := zdalne_wejscia[0].10;
IZ[11] := zdalne_wejscia[0].11;
IZ[12] := zdalne_wejscia[0].12;
IZ[13] := zdalne_wejscia[0].13;
IZ[14] := zdalne_wejscia[0].14;
IZ[15] := zdalne_wejscia[0].15;
END_IF;
END_FUNCTION_BLOCK

(* Visualisation tasmy
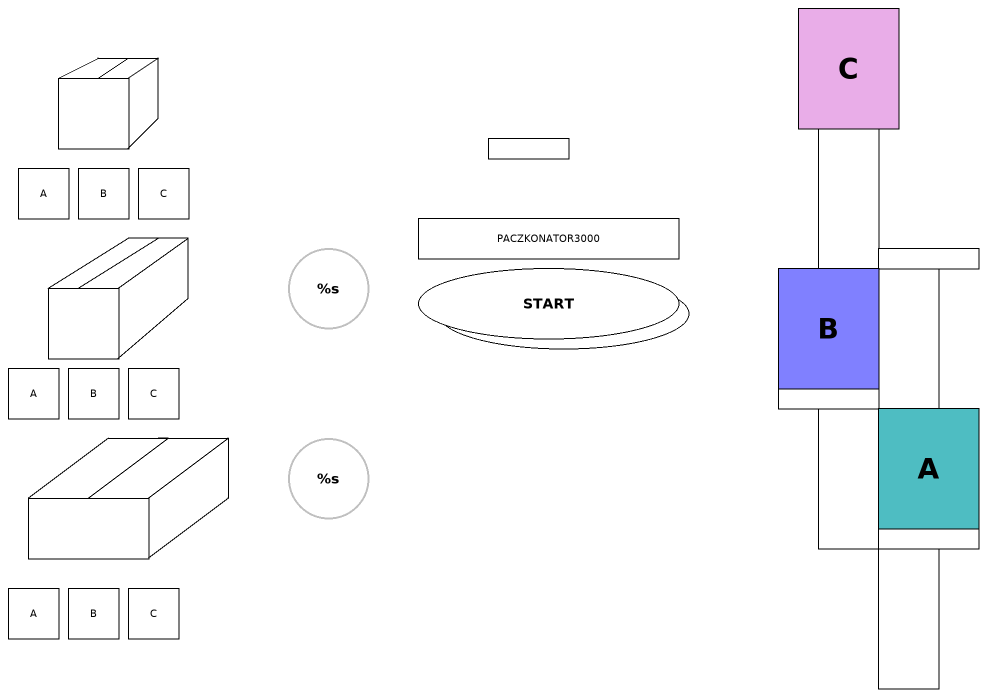
rectangle at (1100,180)-(1161,321): alarm colour if PLC_PRG.qz_4; toggles PLC_PRG.qz_4
rectangle at (1160,320)-(1221,461): alarm colour if PLC_PRG.qz_3; toggles PLC_PRG.qz_3
rectangle at (1100,460)-(1161,601): alarm colour if PLC_PRG.qz_2; toggles PLC_PRG.qz_2
rectangle at (1160,600)-(1221,741): alarm colour if PLC_PRG.qz_1; toggles PLC_PRG.qz_1
rectangle at (1160,580)-(1261,601): shows PLC_PRG.qz_8; alarm colour if PLC_PRG.qz_5; toggles PLC_PRG.qz_5
rectangle at (1060,440)-(1161,461): alarm colour if PLC_PRG.qz_6; toggles PLC_PRG.qz_6
rectangle at (1160,300)-(1261,321): alarm colour if PLC_PRG.qz_7; toggles PLC_PRG.qz_7
rounded rectangle at (1160,460)-(1261,581): text "A"; alarm colour if qz[12]
rounded rectangle at (1060,320)-(1161,441): text "B"; alarm colour if qz[13]
rounded rectangle at (1080,60)-(1181,181): text "C"; alarm colour if qz[11]
rounded rectangle at (290,640)-(341,691): text "A"; alarm colour if PLC_PRG.p1_va; taps PLC_PRG.p1_a
ellipse at (570,300)-(651,381): text "%s"; shows PLC_PRG.size1_count
ellipse at (700,320)-(961,391): text "START"; alarm colour if i2; toggles i2
rounded rectangle at (700,270)-(961,311): text "PACZKONATOR3000"
ellipse at (570,490)-(651,571): text "%s"; shows PLC_PRG.size0_count
rounded rectangle at (350,640)-(401,691): text "B"; alarm colour if PLC_PRG.p1_vb; taps PLC_PRG.p1_b
rounded rectangle at (410,640)-(461,691): text "C"; alarm colour if PLC_PRG.p1_vc; taps PLC_PRG.p1_c
rounded rectangle at (290,420)-(341,471): text "A"; alarm colour if PLC_PRG.p2_va; taps PLC_PRG.p2_a
rounded rectangle at (350,420)-(401,471): text "B"; alarm colour if PLC_PRG.p2_vb; taps PLC_PRG.p2_b
rounded rectangle at (410,420)-(461,471): text "C"; alarm colour if PLC_PRG.p2_vc; taps PLC_PRG.p2_c
rounded rectangle at (300,220)-(351,271): text "A"; alarm colour if PLC_PRG.p3_va; taps PLC_PRG.p3_a
rounded rectangle at (360,220)-(411,271): text "B"; alarm colour if PLC_PRG.p3_vb; taps PLC_PRG.p3_b
rounded rectangle at (420,220)-(471,271): text "C"; alarm colour if PLC_PRG.p3_vc; taps PLC_PRG.p3_c
17 more shapes without text or variables
2 elements of other kinds (tables, trends, ...) not read
*)
